      sync()
    end
  end
  while (True):
    $ 1 "Robot Program"
    $ 2 "MoveJ"
    $ 3 "Apagado" "breakAfter"
    movej(get_inverse_kin(Apagado_p, qnear=Apagado_q), a=1.3962634015954636, v=1.0471975511965976)
    $ 4 "Mantenimiento" "breakAfter"
    movej(get_inverse_kin(Mantenimiento_p, qnear=Mantenimiento_q), a=1.3962634015954636, v=1.0471975511965976)
    $ 5 "Variables"
    $ 6 "muestras≔3"
    global muestras=3
    $ 7 "muestrasTomadas≔0"
    global muestrasTomadas=0
    $ 8 "alpha≔0"
    global alpha=0
    $ 9 "P1≔p[0,0,0,0,0,0]"
    global P1=p[0,0,0,0,0,0]
    $ 10 "P2≔p[0,0,0,0,0,0]"
    global P2=p[0,0,0,0,0,0]
    $ 11 "P3≔p[0,0,0,0,0,0]"
    global P3=p[0,0,0,0,0,0]
    $ 12 "P4≔p[0,0,0,0,0,0]"
    global P4=p[0,0,0,0,0,0]
    $ 13 "Coordenada≔p[0,0,0,0,0,0]"
    global Coordenada=p[0,0,0,0,0,0]
    $ 14 "MoveJ"
    $ 15 "Loop"
    while (True):
      $ 16 "Waypoint_1" "breakAfter"
      movej(get_inverse_kin(Waypoint_1_p, qnear=Waypoint_1_q), a=1.3962634015954636, v=1.0471975511965976)
      $ 17 "Waypoint_2" "breakAfter"
      movej(get_inverse_kin(Waypoint_2_p, qnear=Waypoint_2_q), a=1.3962634015954636, v=1.0471975511965976)
      $ 18 "var_7≔pose_dist(Waypoint_1, Waypoint_2)"
      global var_7= pose_dist (Waypoint_1_p, Waypoint_2_p)
    end
    $ 19 "Waypoint_1" "breakAfter"
    movej(get_inverse_kin(Waypoint_1_p, qnear=Waypoint_1_q), a=1.3962634015954636, v=1.0471975511965976)
    $ 20 "Waypoint_2" "breakAfter"
    movej(get_inverse_kin(Waypoint_2_p, qnear=Waypoint_2_q), a=1.3962634015954636, v=1.0471975511965976)
    $ 21 "pch_atual≔get_actual_tcp_pose()"
    global pch_atual= get_actual_tcp_pose ()
    $ 22 "Popup: hi"
    popup(str_cat("",pch_atual), "Mensaje", False, False, blocking=True)
    $ 23 "Movimiento eje 7"
    $ 24 "MoveL"
    $ 25 "Transporte" "breakAfter"
    movel(Transporte_p, a=1.2, v=0.25)
    $ 26 "Set postrnas_m187=Encender"
    modbus_set_output_signal("postrnas_m187", True)
    $ 28 "num_barreno≔str_cat('Barreno: ',1)"
    global num_barreno=str_cat("Barreno: ",1)
    $ 29 "var_6≔get_actual_tcp_pose()"
    global var_6= get_actual_tcp_pose ()
    $ 30 "X_actual≔str_cat('     X: ',var_6[0])"
    global X_actual=str_cat("     X: ",var_6[0])
    $ 31 "Y_actual≔str_cat('     Y: ',var_6[1])"
    global Y_actual=str_cat("     Y: ",var_6[1])
    $ 32 "pos_barreno≔str_cat(X_actual,Y_actual)"
    global pos_barreno=str_cat(X_actual,Y_actual)
    $ 33 "textmsg('------------------DAS LOG------------------')"
    textmsg("------------------DAS LOG------------------")
    $ 34 "textmsg(num_barreno,pos_barreno)"
    textmsg(num_barreno,pos_barreno)
    $ 35 "Popup: hsjd"
    popup("hsjd", "Advertencia", True, False, blocking=True)
    $ 36 "Saludos"
    $ 37 "MoveL"
    $ 38 "Transporte" "breakAfter"
    movel(Transporte_p, a=1.2, v=0.25)
    $ 39 "Set postrnas_m187=Encender"
    modbus_set_output_signal("postrnas_m187", True)
    $ 42 "MoveJ"
    $ 44 "Set postrnas_m187=Apagar"
    modbus_set_output_signal("postrnas_m187", False)
    $ 45 "Waypoint_3" "breakAfter"
    movej(get_inverse_kin(Waypoint_3_p, qnear=Waypoint_3_q), a=1.3962634015954636, v=1.0471975511965976)
    $ 47 "Loop 15 times"
    Loop_1 = 0
    while (Loop_1 < 15):
      $ 48 "MoveL"
      $ 51 "Waypoint_3" "breakAfter"
      movel(Waypoint_3_p, a=2.2, v=1.5)
      $ 52 "Waypoint_4" "breakAfter"
      movel(Waypoint_4_p, a=2.2, v=1.5)
      Loop_1 = Loop_1 + 1
    end
    $ 57 "Popup: arranquesito"
    popup("arranquesito", "Mensaje", False, False, blocking=True)
    $ 66 "Cambio_Brocas"
    $ 67 "Loop 1 times"
    Loop_1 = 0
    while (Loop_1 < 1):
      $ 68 "MoveJ"
      $ 73 "PreCambio_Broca" "breakAfter"
      movej(get_inverse_kin(PreCambio_Broca_p, qnear=PreCambio_Broca_q), a=1.3962634015954636, v=1.0471975511965976)
      $ 77 "Call Poner_Broca"
      Poner_Broca()
      Loop_1 = Loop_1 + 1
    end
    $ 78 "Barrenado"
    $ 79 "alpha≔0"
    global alpha=0
    $ 80 "Loop"
    while (True):
      $ 81 "MoveJ"
      $ 82 "casa" "breakAfter"
      movej(get_inverse_kin(casa_p, qnear=casa_q), a=1.3962634015954636, v=1.0471975511965976)
      $ 83 "Call Calibracion"
      Calibracion()
      $ 84 "Call GoNoGo"
      GoNoGo()
      $ 85 "MoveL"
      $ 86 "Barreno1" "breakAfter"
      movel(Barreno1_p, a=1.2, v=0.25)
      $ 87 "Barreno2" "breakAfter"
      movel(Barreno2_p, a=1.2, v=0.25)
      $ 88 "Loop 2 times"
      Loop_9 = 0
      while (Loop_9 < 2):
        $ 89 "If alpha≤16"
        if (alpha <= 16):
          $ 90 "internos≔interpolate_pose(Barreno1, Barreno2, alpha)"
          global internos= interpolate_pose (Barreno1_p, Barreno2_p, alpha)
          $ 91 "bajada≔p[0,0,-0.024,0,0,0]"
          global bajada=p[0,0,-0.024,0,0,0]
          $ 92 "subida≔p[0,0,0.024,0,0,0]"
          global subida=p[0,0,0.024,0,0,0]
          $ 93 "internos" "breakAfter"
          movel(internos, a=1.2, v=0.25)
          $ 94 "Direction: Base Z-"
          global move_thread_flag_94=0
          thread move_thread_94():
            enter_critical
            move_thread_flag_94 = 1
            local towardsPos=calculate_point_to_move_towards(p[0.0,0.0,0.0,0.0,0.0,0.0], [0.0,0.0,-1.0], 0.067)
            movel(towardsPos, a=1.2, v=0.25)
            move_thread_flag_94 = 2
            exit_critical
          end
          move_thread_flag_94 = 0
          move_thread_han_94 = run move_thread_94()
          while (True):
            sleep(1.0E-10)
            if (move_thread_flag_94 > 1):
              join move_thread_han_94
              $ 95 "Until (distance)"
              break
            end
            sync()
          end
          $ 96 "Direction: Base Z-"
          global move_thread_flag_96=0
          thread move_thread_96():
            enter_critical
            move_thread_flag_96 = 1
            local towardsPos=calculate_point_to_move_towards(p[0.0,0.0,0.0,0.0,0.0,0.0], [0.0,0.0,-1.0], 1000.0)
            movel(towardsPos, a=2.0E-4, v=0.0013)
            move_thread_flag_96 = 2
            exit_critical
          end
          move_thread_flag_96 = 0
          move_thread_han_96 = run move_thread_96()
          while (True):
            local targetTcpDirection=get_target_tcp_speed()
            local stepsToRetract=tool_contact(direction=targetTcpDirection)
            if (stepsToRetract > 0):
              kill move_thread_han_96
              stopl(9.0)
              local backTrackMovement=get_actual_joint_positions_history(stepsToRetract)
              local contactPose=get_forward_kin(backTrackMovement)
              local posDir=[targetTcpDirection[0],targetTcpDirection[1],targetTcpDirection[2]]
              local retractTo=contactPose
              if (norm(posDir) > 1e-6):
                local normalizedPosDir=normalize(posDir)
                local additionalRetraction=p[normalizedPosDir[0] * 0.0, normalizedPosDir[1] * 0.0, normalizedPosDir[2] * 0.0, 0, 0, 0]
                retractTo = pose_sub(contactPose, additionalRetraction)
              end
              movel(retractTo, a=9.0, v=0.1)
              $ 97 "Until (tool_contact_detection)"
              break
            end
            sync()
          end
          $ 98 "Wait: 0.3"
          sleep(0.3)
          $ 99 "Set CO[1]=Encender"
          set_configurable_digital_out(1, True)
          $ 100 "Wait: 0.5"
          sleep(0.5)
          $ 101 "Set CO[1]=Apagar"
          set_configurable_digital_out(1, False)
          $ 102 "Direction: Base Z+"
          global move_thread_flag_102=0
          thread move_thread_102():
            enter_critical
            move_thread_flag_102 = 1
            local towardsPos=calculate_point_to_move_towards(p[0.0,0.0,0.0,0.0,0.0,0.0], [0.0,0.0,1.0], 0.002)
            movel(towardsPos, a=1.2, v=0.25)
            move_thread_flag_102 = 2
            exit_critical
          end
          move_thread_flag_102 = 0
          move_thread_han_102 = run move_thread_102()
          while (True):
            sleep(1.0E-10)
            if (move_thread_flag_102 > 1):
              join move_thread_han_102
              $ 103 "Until (distance)"
              break
            end
            sync()
          end
          $ 104 "Wait: 0.5"
          sleep(0.5)
          $ 105 "Set CO[1]=Encender"
          set_configurable_digital_out(1, True)
          $ 106 "Wait: 0.3"
          sleep(0.3)
          $ 107 "Loop 1 times"
          Loop_6 = 0
          while (Loop_6 < 1):
            $ 108 "bajar≔pose_add(get_actual_tcp_pose(), bajada)"
            global bajar= pose_add ( get_actual_tcp_pose (), bajada)
            $ 109 "bajar" "breakAfter"
            movel(bajar, a=0.01, v=0.005)
            $ 110 "subir≔pose_add(get_actual_tcp_pose(), subida)"
            global subir= pose_add ( get_actual_tcp_pose (), subida)
            $ 111 "subir" "breakAfter"
            movel(subir, a=0.02, v=0.02)
            $ 112 "bajada≔pose_add(bajada, p[0,0,-0.008,0,0,0])"
            global bajada= pose_add (bajada, p[0,0,-0.008,0,0,0])
            $ 113 "subida≔pose_add(subida, p[0,0,0.008,0,0,0])"
            global subida= pose_add (subida, p[0,0,0.008,0,0,0])
            Loop_6 = Loop_6 + 1
          end
          $ 114 "Set CO[1]=Apagar"
          set_configurable_digital_out(1, False)
          $ 115 "Direction: Base Z+"
          global move_thread_flag_115=0
          thread move_thread_115():
            enter_critical
            move_thread_flag_115 = 1
            local towardsPos=calculate_point_to_move_towards(p[0.0,0.0,0.0,0.0,0.0,0.0], [0.0,0.0,1.0], 0.1)
            movel(towardsPos, a=1.2, v=0.25)
            move_thread_flag_115 = 2
            exit_critical
          end
          move_thread_flag_115 = 0
          move_thread_han_115 = run move_thread_115()
          while (True):
            sleep(1.0E-10)
            if (move_thread_flag_115 > 1):
              join move_thread_han_115
              $ 116 "Until (distance)"
              break
            end
            sync()
          end
          $ 117 "alpha≔alpha+1"
          global alpha=alpha+1
        else:
          $ 118 "Else" "noBreak"
          $ 119 "Popup: linea barrenada"
          popup("linea barrenada", "Mensaje", False, False, blocking=True)
          $ 120 "Call Quitar_Broca_Chida"
          Quitar_Broca_Chida()
          $ 121 "Popup: fin"
          popup("fin", "Mensaje", False, False, blocking=True)
        end
        Loop_9 = Loop_9 + 1
      end
      $ 122 "Call Quitar_Broca_Chida"
      Quitar_Broca_Chida()
      $ 123 "Call Poner_Broca"
      Poner_Broca()
    end
  end
end
